ABB RAPID module: Module1.mod

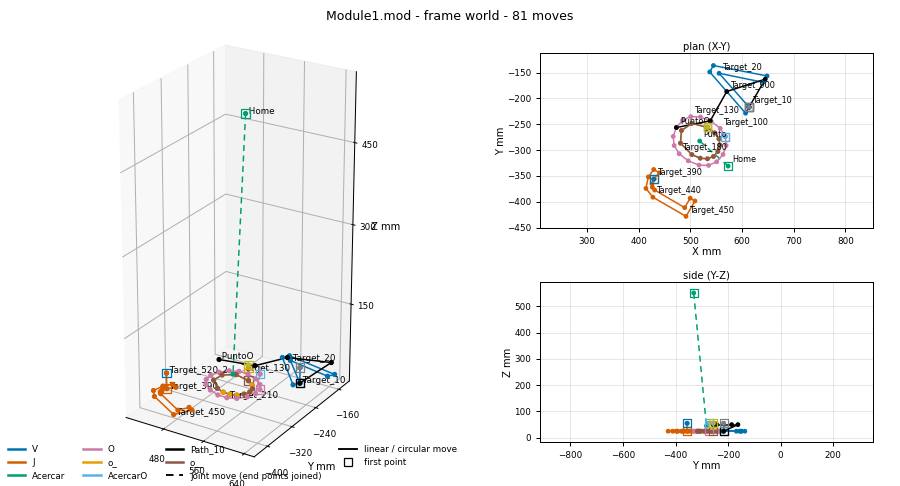
[picture p0: tool path of Module1.mod in frame world, 81 of 82 moves have a stored position in this frame; points joined in program order, loops and branches not executed]
MODULE Module1
        CONST robtarget Target_10:=[[139.847323193,319.022708542,15],[0,0.707106781,0.707106781,0],[0,0,0,0],[9E+09,9E+09,9E+09,9E+09,9E+09,9E+09]];
    CONST robtarget Target_20:=[[56.784114117,346.737457327,15],[0,0.707106781,0.707106781,0],[0,0,0,0],[9E+09,9E+09,9E+09,9E+09,9E+09,9E+09]];
    CONST robtarget Target_30:=[[139.847323193,374.452206111,15],[0,0.707106781,0.707106781,0],[0,0,0,0],[9E+09,9E+09,9E+09,9E+09,9E+09,9E+09]];
    CONST robtarget Target_40:=[[139.847323193,388.714766889,15],[0,0.707106781,0.707106781,0],[0,0,0,0],[9E+09,9E+09,9E+09,9E+09,9E+09,9E+09]];
    CONST robtarget Target_50:=[[39.847323193,354.273924101,15],[0,0.707106781,0.707106781,0],[0,0,0,0],[9E+09,9E+09,9E+09,9E+09,9E+09,9E+09]];
    CONST robtarget Target_60:=[[39.847323193,339.930326046,15],[0,0.707106781,0.707106781,0],[0,0,0,0],[9E+09,9E+09,9E+09,9E+09,9E+09,9E+09]];
    CONST robtarget Target_70:=[[139.847323193,305.489483258,15],[0,0.707106781,0.707106781,0],[0,0,0,0],[9E+09,9E+09,9E+09,9E+09,9E+09,9E+09]];
    CONST robtarget Target_80:=[[139.847323193,319.022708542,15],[0,0.707106781,0.707106781,0],[0,0,0,0],[9E+09,9E+09,9E+09,9E+09,9E+09,9E+09]];
    CONST robtarget Target_90:=[[128.421067116,246.656420049,15],[0,0.707106781,0.707106781,0],[0,0,0,0],[9E+09,9E+09,9E+09,9E+09,9E+09,9E+09]];
    CONST robtarget Target_100:=[[111.970499855,255.530001897,15],[0,0.707106781,0.707106781,0],[0,0,0,0],[9E+09,9E+09,9E+09,9E+09,9E+09,9E+09]];
    CONST robtarget Target_110:=[[89.847323193,258.649937067,15],[0,0.707106781,0.707106781,0],[0,0,0,0],[9E+09,9E+09,9E+09,9E+09,9E+09,9E+09]];
    CONST robtarget Target_120:=[[67.764665171,255.570520536,15],[0,0.707106781,0.707106781,0],[0,0,0,0],[9E+09,9E+09,9E+09,9E+09,9E+09,9E+09]];
    CONST robtarget Target_130:=[[51.354616548,246.737457327,15],[0,0.707106781,0.707106781,0],[0,0,0,0],[9E+09,9E+09,9E+09,9E+09,9E+09,9E+09]];
    CONST robtarget Target_140:=[[41.184438266,232.71800838,15],[0,0.707106781,0.707106781,0],[0,0,0,0],[9E+09,9E+09,9E+09,9E+09,9E+09,9E+09]];
    CONST robtarget Target_150:=[[37.740353988,214.484621022,15],[0,0.707106781,0.707106781,0],[0,0,0,0],[9E+09,9E+09,9E+09,9E+09,9E+09,9E+09]];
    CONST robtarget Target_460:=[[139.847323193,109.460309839,15],[0,0.707106781,0.707106781,0],[0,0,0,0],[9E+09,9E+09,9E+09,9E+09,9E+09,9E+09]];
    CONST robtarget Target_470:=[[129.231439887,109.460309839,15],[0,0.707106781,0.707106781,0],[0,0,0,0],[9E+09,9E+09,9E+09,9E+09,9E+09,9E+09]];
    CONST robtarget Target_480:=[[129.231439887,88.309580503,15],[0,0.707106781,0.707106781,0],[0,0,0,0],[9E+09,9E+09,9E+09,9E+09,9E+09,9E+09]];
    CONST robtarget Target_490:=[[61.970499855,88.795804166,15],[0,0.707106781,0.707106781,0],[0,0,0,0],[9E+09,9E+09,9E+09,9E+09,9E+09,9E+09]];
    CONST robtarget Target_500:=[[55.406480406,91.145885203,15],[0,0.707106781,0.707106781,0],[0,0,0,0],[9E+09,9E+09,9E+09,9E+09,9E+09,9E+09]];
    CONST robtarget Target_510:=[[51.395135187,96.534864134,15],[0,0.707106781,0.707106781,0],[0,0,0,0],[9E+09,9E+09,9E+09,9E+09,9E+09,9E+09]];
    CONST robtarget Target_520:=[[49.976982837,106.380893307,15],[0,0.707106781,0.707106781,0],[0,0,0,0],[9E+09,9E+09,9E+09,9E+09,9E+09,9E+09]];
    CONST robtarget Target_530:=[[129.231439887,88.309580503,15],[0,1,0,0],[0,0,0,0],[9E+09,9E+09,9E+09,9E+09,9E+09,9E+09]];
    CONST robtarget Target_540:=[[61.970499855,88.795804166,15],[0,1,0,0],[0,0,0,0],[9E+09,9E+09,9E+09,9E+09,9E+09,9E+09]];
    CONST robtarget Target_550:=[[55.406480406,91.145885203,15],[0,1,0,0],[0,0,0,0],[9E+09,9E+09,9E+09,9E+09,9E+09,9E+09]];
    CONST robtarget Target_560:=[[51.395135187,96.534864134,15],[0,1,0,0],[0,0,0,0],[9E+09,9E+09,9E+09,9E+09,9E+09,9E+09]];
    CONST robtarget Target_570:=[[49.976982837,106.380893307,15],[0,1,0,0],[0,0,0,0],[9E+09,9E+09,9E+09,9E+09,9E+09,9E+09]];
    CONST robtarget Target_580:=[[53.218473923,122.264199628,15],[0,1,0,0],[0,0,0,0],[9E+09,9E+09,9E+09,9E+09,9E+09,9E+09]];
    CONST robtarget Target_590:=[[40.414584134,122.264199628,15],[0,1,0,0],[0,0,0,0],[9E+09,9E+09,9E+09,9E+09,9E+09,9E+09]];
    CONST robtarget Home:=[[161.779515601,200,541.048881024],[0.5,0,0.866025404,0],[0,0,0,0],[9E+09,9E+09,9E+09,9E+09,9E+09,9E+09]];
    CONST robtarget Punto:=[[89.89,214.443,35],[0,1,0,0],[0,0,-2,0],[9E+09,9E+09,9E+09,9E+09,9E+09,9E+09]];
    CONST robtarget Target_600:=[[37.740353988,214.484621022,15],[0,1,0,0],[0,0,0,0],[9E+09,9E+09,9E+09,9E+09,9E+09,9E+09]];
    CONST robtarget Target_610:=[[41.062882351,196.534864134,15],[0,1,0,0],[0,0,0,0],[9E+09,9E+09,9E+09,9E+09,9E+09,9E+09]];
    CONST robtarget Target_620:=[[51.354616548,182.231784717,15],[0,1,0,0],[0,0,0,0],[9E+09,9E+09,9E+09,9E+09,9E+09,9E+09]];
    CONST robtarget Target_630:=[[67.845702448,173.317684231,15],[0,1,0,0],[0,0,0,0],[9E+09,9E+09,9E+09,9E+09,9E+09,9E+09]];
    CONST robtarget Target_640:=[[89.847323193,170.238267699,15],[0,1,0,0],[0,0,0,0],[9E+09,9E+09,9E+09,9E+09,9E+09,9E+09]];
    CONST robtarget Target_650:=[[112.051537132,173.398721508,15],[0,1,0,0],[0,0,0,0],[9E+09,9E+09,9E+09,9E+09,9E+09,9E+09]];
    CONST robtarget Target_660:=[[128.421067116,182.231784717,15],[0,1,0,0],[0,0,0,0],[9E+09,9E+09,9E+09,9E+09,9E+09,9E+09]];
    CONST robtarget Target_670:=[[138.388652205,196.089159109,15],[0,1,0,0],[0,0,0,0],[9E+09,9E+09,9E+09,9E+09,9E+09,9E+09]];
    CONST robtarget Target_680:=[[141.954292399,214.484621022,15],[0,1,0,0],[0,0,0,0],[9E+09,9E+09,9E+09,9E+09,9E+09,9E+09]];
    CONST robtarget Target_690:=[[138.510208121,232.677489741,15],[0,1,0,0],[0,0,0,0],[9E+09,9E+09,9E+09,9E+09,9E+09,9E+09]];
    CONST robtarget Target_700:=[[128.421067116,246.656420049,15],[0,1,0,0],[0,0,0,0],[9E+09,9E+09,9E+09,9E+09,9E+09,9E+09]];
    CONST robtarget Target_710:=[[111.970499855,255.530001897,15],[0,1,0,0],[0,0,0,0],[9E+09,9E+09,9E+09,9E+09,9E+09,9E+09]];
    CONST robtarget Target_720:=[[89.847323193,258.649937067,15],[0,1,0,0],[0,0,0,0],[9E+09,9E+09,9E+09,9E+09,9E+09,9E+09]];
    CONST robtarget Target_730:=[[67.764665171,255.570520536,15],[0,1,0,0],[0,0,0,0],[9E+09,9E+09,9E+09,9E+09,9E+09,9E+09]];
    CONST robtarget Target_740:=[[51.354616548,246.737457327,15],[0,1,0,0],[0,0,0,0],[9E+09,9E+09,9E+09,9E+09,9E+09,9E+09]];
    CONST robtarget Target_750:=[[41.184438266,232.71800838,15],[0,1,0,0],[0,0,0,0],[9E+09,9E+09,9E+09,9E+09,9E+09,9E+09]];
    CONST robtarget Target_760:=[[37.740353988,214.484621022,15],[0,1,0,0],[0,0,0,0],[9E+09,9E+09,9E+09,9E+09,9E+09,9E+09]];
    CONST robtarget Target_770:=[[89.847323193,244.792562675,15],[0,1,0,0],[0,0,0,0],[9E+09,9E+09,9E+09,9E+09,9E+09,9E+09]];
    CONST robtarget Target_780:=[[107.27033778,242.685593469,15],[0,1,0,0],[0,0,0,0],[9E+09,9E+09,9E+09,9E+09,9E+09,9E+09]];
    CONST robtarget Target_790:=[[120.074227569,236.607797683,15],[0,1,0,0],[0,0,0,0],[9E+09,9E+09,9E+09,9E+09,9E+09,9E+09]];
    CONST robtarget Target_800:=[[127.934843453,227.04539898,15],[0,1,0,0],[0,0,0,0],[9E+09,9E+09,9E+09,9E+09,9E+09,9E+09]];
    CONST robtarget Target_810:=[[130.446999044,214.403583745,15],[0,1,0,0],[0,0,0,0],[9E+09,9E+09,9E+09,9E+09,9E+09,9E+09]];
    CONST robtarget Target_820:=[[127.853806176,201.842805787,15],[0,1,0,0],[0,0,0,0],[9E+09,9E+09,9E+09,9E+09,9E+09,9E+09]];
    CONST robtarget Target_830:=[[120.074227569,192.280407083,15],[0,1,0,0],[0,0,0,0],[9E+09,9E+09,9E+09,9E+09,9E+09,9E+09]];
    CONST robtarget Target_840:=[[107.391893696,186.243129936,15],[0,1,0,0],[0,0,0,0],[9E+09,9E+09,9E+09,9E+09,9E+09,9E+09]];
    CONST robtarget Target_850:=[[89.847323193,184.095642092,15],[0,1,0,0],[0,0,0,0],[9E+09,9E+09,9E+09,9E+09,9E+09,9E+09]];
    CONST robtarget Target_860:=[[59.701456095,192.320925722,15],[0,1,0,0],[0,0,0,0],[9E+09,9E+09,9E+09,9E+09,9E+09,9E+09]];
    CONST robtarget Target_870:=[[49.247647343,214.403583745,15],[0,1,0,0],[0,0,0,0],[9E+09,9E+09,9E+09,9E+09,9E+09,9E+09]];
    CONST robtarget Target_880:=[[59.701456095,236.526760406,15],[0,1,0,0],[0,0,0,0],[9E+09,9E+09,9E+09,9E+09,9E+09,9E+09]];
    CONST robtarget Target_890:=[[89.847323193,244.792562675,15],[0,1,0,0],[0,0,0,0],[9E+09,9E+09,9E+09,9E+09,9E+09,9E+09]];
    CONST robtarget puntoV:=[[139.847,381.583,40],[0,1,0,0],[0,0,-2,0],[9E+09,9E+09,9E+09,9E+09,9E+09,9E+09]];
    CONST robtarget puntoV_2:=[[139.847,381.583,40],[0,1,0,0],[0,0,-2,0],[9E+09,9E+09,9E+09,9E+09,9E+09,9E+09]];
    CONST robtarget puntoJ_2:=[[40.415,122.264,40],[0,1,0,0],[-1,0,1,0],[9E+09,9E+09,9E+09,9E+09,9E+09,9E+09]];
    CONST robtarget puntoJ:=[[40.415,122.264,40],[0,1,0,0],[-1,0,1,0],[9E+09,9E+09,9E+09,9E+09,9E+09,9E+09]];
    CONST robtarget PuntoO_2:=[[37.74,214.485,40],[0,1,0,0],[0,0,0,0],[9E+09,9E+09,9E+09,9E+09,9E+09,9E+09]];
    CONST robtarget PuntoO:=[[37.740005074,214.485004022,40.000022651],[0,1,0,0],[0,0,-2,0],[9E+09,9E+09,9E+09,9E+09,9E+09,9E+09]];
    CONST robtarget punto_opeq_2:=[[89.847,244.793,40],[0,1,0,0],[0,0,0,0],[9E+09,9E+09,9E+09,9E+09,9E+09,9E+09]];
    CONST robtarget punto_opeq:=[[89.847,244.793,40],[0,1,0,0],[0,0,0,0],[9E+09,9E+09,9E+09,9E+09,9E+09,9E+09]];
    CONST robtarget Target_900:=[[87.275,323.596,40],[0,1,0,0],[0,0,-2,0],[9E+09,9E+09,9E+09,9E+09,9E+09,9E+09]];
    CONST robtarget Target_910:=[[88.022,258.633,40],[0,1,0,0],[0,0,-2,0],[9E+09,9E+09,9E+09,9E+09,9E+09,9E+09]];
    CONST robtarget Target_80_2:=[[139.847323193,319.022708542,45],[0,0.707106781,0.707106781,0],[0,0,1,0],[9E+09,9E+09,9E+09,9E+09,9E+09,9E+09]];
    CONST robtarget Target_160:=[[41.062882351,196.534864134,15],[0,0.707106781,0.707106781,0],[0,0,0,0],[9E+09,9E+09,9E+09,9E+09,9E+09,9E+09]];
    CONST robtarget Target_230:=[[141.954292399,214.484621022,15],[0,0.707106781,0.707106781,0],[0,0,0,0],[9E+09,9E+09,9E+09,9E+09,9E+09,9E+09]];
    CONST robtarget Target_180:=[[67.845702448,173.317684231,15],[0,0.707106781,0.707106781,0],[0,0,0,0],[9E+09,9E+09,9E+09,9E+09,9E+09,9E+09]];
    CONST robtarget Target_240:=[[138.510208121,232.677489741,15],[0,0.707106781,0.707106781,0],[0,0,0,0],[9E+09,9E+09,9E+09,9E+09,9E+09,9E+09]];
    CONST robtarget Target_200:=[[112.051537132,173.398721508,15],[0,0.707106781,0.707106781,0],[0,0,0,0],[9E+09,9E+09,9E+09,9E+09,9E+09,9E+09]];
    CONST robtarget Target_220:=[[138.388652205,196.089159109,15],[0,0.707106781,0.707106781,0],[0,0,0,0],[9E+09,9E+09,9E+09,9E+09,9E+09,9E+09]];
    CONST robtarget Target_170:=[[51.354616548,182.231784717,15],[0,0.707106781,0.707106781,0],[0,0,0,0],[9E+09,9E+09,9E+09,9E+09,9E+09,9E+09]];
    CONST robtarget Target_210:=[[128.421067116,182.231784717,15],[0,0.707106781,0.707106781,0],[0,0,0,0],[9E+09,9E+09,9E+09,9E+09,9E+09,9E+09]];
    CONST robtarget Target_190:=[[89.847323193,170.238267699,15],[0,0.707106781,0.707106781,0],[0,0,0,0],[9E+09,9E+09,9E+09,9E+09,9E+09,9E+09]];
    CONST robtarget Target_250_2:=[[128.421067116,246.656420049,45],[0,0.707106781,0.707106781,0],[0,0,1,0],[9E+09,9E+09,9E+09,9E+09,9E+09,9E+09]];
    CONST robtarget Target_260:=[[89.847323193,244.792562675,15],[0,0.707106781,0.707106781,0],[0,0,0,0],[9E+09,9E+09,9E+09,9E+09,9E+09,9E+09]];
    CONST robtarget Target_270:=[[107.27033778,242.685593469,15],[0,0.707106781,0.707106781,0],[0,0,0,0],[9E+09,9E+09,9E+09,9E+09,9E+09,9E+09]];
    CONST robtarget Target_280:=[[120.074227569,236.607797683,15],[0,0.707106781,0.707106781,0],[0,0,0,0],[9E+09,9E+09,9E+09,9E+09,9E+09,9E+09]];
    CONST robtarget Target_290:=[[127.934843453,227.04539898,15],[0,0.707106781,0.707106781,0],[0,0,0,0],[9E+09,9E+09,9E+09,9E+09,9E+09,9E+09]];
    CONST robtarget Target_300:=[[130.446999044,214.403583745,15],[0,0.707106781,0.707106781,0],[0,0,0,0],[9E+09,9E+09,9E+09,9E+09,9E+09,9E+09]];
    CONST robtarget Target_310:=[[127.853806176,201.842805787,15],[0,0.707106781,0.707106781,0],[0,0,0,0],[9E+09,9E+09,9E+09,9E+09,9E+09,9E+09]];
    CONST robtarget Target_320:=[[120.074227569,192.280407083,15],[0,0.707106781,0.707106781,0],[0,0,0,0],[9E+09,9E+09,9E+09,9E+09,9E+09,9E+09]];
    CONST robtarget Target_330:=[[107.391893696,186.243129936,15],[0,0.707106781,0.707106781,0],[0,0,0,0],[9E+09,9E+09,9E+09,9E+09,9E+09,9E+09]];
    CONST robtarget Target_340:=[[89.847323193,184.095642092,15],[0,0.707106781,0.707106781,0],[0,0,0,0],[9E+09,9E+09,9E+09,9E+09,9E+09,9E+09]];
    CONST robtarget Target_350:=[[59.701456095,192.320925722,15],[0,0.707106781,0.707106781,0],[0,0,0,0],[9E+09,9E+09,9E+09,9E+09,9E+09,9E+09]];
    CONST robtarget Target_360:=[[49.247647343,214.403583745,15],[0,0.707106781,0.707106781,0],[0,0,0,0],[9E+09,9E+09,9E+09,9E+09,9E+09,9E+09]];
    CONST robtarget Target_370:=[[59.701456095,236.526760406,15],[0,0.707106781,0.707106781,0],[0,0,0,0],[9E+09,9E+09,9E+09,9E+09,9E+09,9E+09]];
    CONST robtarget Target_380:=[[89.847323193,244.792562675,15],[0,0.707106781,0.707106781,0],[0,0,0,0],[9E+09,9E+09,9E+09,9E+09,9E+09,9E+09]];
    CONST robtarget Target_380_2:=[[89.847323193,244.792562675,45],[0,0.707106781,0.707106781,0],[0,0,1,0],[9E+09,9E+09,9E+09,9E+09,9E+09,9E+09]];
    CONST robtarget Target_520_2:=[[49.976982837,106.380893307,45],[0,0.707106781,0.707106781,0],[0,0,0,0],[9E+09,9E+09,9E+09,9E+09,9E+09,9E+09]];
    CONST robtarget Target_410:=[[40.414584134,122.264199628,15],[0,0.707106781,0.707106781,0],[0,0,0,0],[9E+09,9E+09,9E+09,9E+09,9E+09,9E+09]];
    CONST robtarget Target_400:=[[53.218473923,122.264199628,15],[0,0.707106781,0.707106781,0],[0,0,0,0],[9E+09,9E+09,9E+09,9E+09,9E+09,9E+09]];
    CONST robtarget Target_390:=[[49.976982837,106.380893307,15],[0,0.707106781,0.707106781,0],[0,0,0,0],[9E+09,9E+09,9E+09,9E+09,9E+09,9E+09]];
    CONST robtarget Target_440:=[[65.860289158,75.019467051,15],[0,0.707106781,0.707106781,0],[0,0,0,0],[9E+09,9E+09,9E+09,9E+09,9E+09,9E+09]];
    CONST robtarget Target_420:=[[38.469689482,104.59807321,15],[0,0.707106781,0.707106781,0],[0,0,0,0],[9E+09,9E+09,9E+09,9E+09,9E+09,9E+09]];
    CONST robtarget Target_430:=[[45.600969871,83.042157489,15],[0,0.707106781,0.707106781,0],[0,0,0,0],[9E+09,9E+09,9E+09,9E+09,9E+09,9E+09]];
    CONST robtarget Target_450:=[[139.847323193,75.019467051,15],[0,0.707106781,0.707106781,0],[0,0,0,0],[9E+09,9E+09,9E+09,9E+09,9E+09,9E+09]];
    CONST jointtarget home2:=[[0,0,0,0,0,0],[9E+09,9E+09,9E+09,9E+09,9E+09,9E+09]];
!***********************************************************
    !
    ! Module:  Module1
    !
    ! Description:
    !   <Insert description here>
    !
    ! Author: Valentina Cruz DP
    !
    ! Version: 1.0
    !
    !***********************************************************


    !***********************************************************
    !
    ! Procedure main
    !
    !   This is the entry point of your program
    !
    !***********************************************************
    PROC main()

     homee;
     AcercarV;
     V;
     AcercarO;
     O;
     AcercarO_;
     o__;
     AcercarJ;
     J;
     homee;

    ENDPROC
    PROC V()
        MoveL Target_10,v60,z1,HerramientaVOJ\WObj:=WorkobjectVOJ;
        MoveL Target_20,v60,z1,HerramientaVOJ\WObj:=WorkobjectVOJ;
        MoveL Target_30,v60,z1,HerramientaVOJ\WObj:=WorkobjectVOJ;
        MoveL Target_40,v60,z1,HerramientaVOJ\WObj:=WorkobjectVOJ;
        MoveL Target_50,v60,z1,HerramientaVOJ\WObj:=WorkobjectVOJ;
        MoveL Target_60,v60,z1,HerramientaVOJ\WObj:=WorkobjectVOJ;
        MoveL Target_70,v60,z1,HerramientaVOJ\WObj:=WorkobjectVOJ;
        MoveL Target_80,v60,z1,HerramientaVOJ\WObj:=WorkobjectVOJ;
        MoveL Target_80_2,v60,z1,HerramientaVOJ\WObj:=WorkobjectVOJ;
    ENDPROC
    PROC J()
        MoveL Target_390,v60,z1,HerramientaVOJ\WObj:=WorkobjectVOJ;
        MoveL Target_400,v60,z1,HerramientaVOJ\WObj:=WorkobjectVOJ;
        MoveL Target_410,v60,z1,HerramientaVOJ\WObj:=WorkobjectVOJ;
        MoveL Target_420,v60,z1,HerramientaVOJ\WObj:=WorkobjectVOJ;
        MoveL Target_430,v60,z1,HerramientaVOJ\WObj:=WorkobjectVOJ;
        MoveL Target_440,v60,z1,HerramientaVOJ\WObj:=WorkobjectVOJ;
        MoveL Target_450,v60,z1,HerramientaVOJ\WObj:=WorkobjectVOJ;
        MoveL Target_460,v60,z1,HerramientaVOJ\WObj:=WorkobjectVOJ;
        MoveL Target_470,v60,z1,HerramientaVOJ\WObj:=WorkobjectVOJ;
        MoveL Target_480,v60,z1,HerramientaVOJ\WObj:=WorkobjectVOJ;
        MoveL Target_490,v60,z1,HerramientaVOJ\WObj:=WorkobjectVOJ;
        MoveL Target_500,v60,z1,HerramientaVOJ\WObj:=WorkobjectVOJ;
        MoveL Target_510,v60,z1,HerramientaVOJ\WObj:=WorkobjectVOJ;
        MoveL Target_520,v60,z1,HerramientaVOJ\WObj:=WorkobjectVOJ;
        MoveL Target_520_2,v60,z1,HerramientaVOJ\WObj:=WorkobjectVOJ;
    ENDPROC
    PROC Acercar()
        MoveJ Home,v200,z1,HerramientaVOJ\WObj:=WorkobjectVOJ;
        MoveJ Punto,v200,z1,HerramientaVOJ\WObj:=WorkobjectVOJ;
    ENDPROC
    PROC Alejar()
    ENDPROC
    PROC O()
        MoveL Target_90,v60,z1,HerramientaVOJ\WObj:=WorkobjectVOJ;
        MoveL Target_100,v60,z1,HerramientaVOJ\WObj:=WorkobjectVOJ;
        MoveL Target_110,v60,z1,HerramientaVOJ\WObj:=WorkobjectVOJ;
        MoveL Target_120,v60,z1,HerramientaVOJ\WObj:=WorkobjectVOJ;
        MoveL Target_130,v60,z1,HerramientaVOJ\WObj:=WorkobjectVOJ;
        MoveL Target_140,v60,z1,HerramientaVOJ\WObj:=WorkobjectVOJ;
        MoveL Target_150,v60,z1,HerramientaVOJ\WObj:=WorkobjectVOJ;
        MoveL Target_160,v60,z1,HerramientaVOJ\WObj:=WorkobjectVOJ;
        MoveL Target_170,v60,z1,HerramientaVOJ\WObj:=WorkobjectVOJ;
        MoveL Target_180,v60,z1,HerramientaVOJ\WObj:=WorkobjectVOJ;
        MoveL Target_190,v60,z1,HerramientaVOJ\WObj:=WorkobjectVOJ;
        MoveL Target_200,v60,z1,HerramientaVOJ\WObj:=WorkobjectVOJ;
        MoveL Target_210,v60,z1,HerramientaVOJ\WObj:=WorkobjectVOJ;
        MoveL Target_220,v60,z1,HerramientaVOJ\WObj:=WorkobjectVOJ;
        MoveL Target_230,v60,z1,HerramientaVOJ\WObj:=WorkobjectVOJ;
        MoveL Target_240,v60,z1,HerramientaVOJ\WObj:=WorkobjectVOJ;
        MoveL Target_250_2,v60,z1,HerramientaVOJ\WObj:=WorkobjectVOJ;
    ENDPROC
    PROC o_()
        MoveL punto_opeq_2,v60,z1,HerramientaVOJ\WObj:=WorkobjectVOJ;
        MoveL Target_770,v60,z1,HerramientaVOJ\WObj:=WorkobjectVOJ;
        MoveL Target_780,v60,z1,HerramientaVOJ\WObj:=WorkobjectVOJ;
        MoveL Target_790,v60,z1,HerramientaVOJ\WObj:=WorkobjectVOJ;
        MoveL Target_800,v60,z1,HerramientaVOJ\WObj:=WorkobjectVOJ;
        MoveL Target_810,v60,z1,HerramientaVOJ\WObj:=WorkobjectVOJ;
        MoveL Target_820,v60,z1,HerramientaVOJ\WObj:=WorkobjectVOJ;
        MoveL Target_830,v60,z1,HerramientaVOJ\WObj:=WorkobjectVOJ;
        MoveL Target_840,v60,z1,HerramientaVOJ\WObj:=WorkobjectVOJ;
        MoveL Target_850,v60,z1,HerramientaVOJ\WObj:=WorkobjectVOJ;
        MoveL Target_860,v60,z1,HerramientaVOJ\WObj:=WorkobjectVOJ;
        MoveL Target_870,v60,z1,HerramientaVOJ\WObj:=WorkobjectVOJ;
        MoveL Target_880,v60,z1,HerramientaVOJ\WObj:=WorkobjectVOJ;
        MoveL Target_890,v60,z1,HerramientaVOJ\WObj:=WorkobjectVOJ;
        MoveL punto_opeq,v60,z1,HerramientaVOJ\WObj:=WorkobjectVOJ;
    ENDPROC
    PROC AcercarO()
        MoveJ Target_250_2,v60,z1,HerramientaVOJ\WObj:=WorkobjectVOJ;
    ENDPROC
    PROC Path_10()
        MoveL Target_10,v200,z1,HerramientaVOJ\WObj:=WorkobjectVOJ;
        MoveL puntoV,v200,z1,HerramientaVOJ\WObj:=WorkobjectVOJ;
        MoveL Target_900,v200,z1,HerramientaVOJ\WObj:=WorkobjectVOJ;
        MoveL Target_910,v200,z1,HerramientaVOJ\WObj:=WorkobjectVOJ;
        MoveL PuntoO,v200,z1,HerramientaVOJ\WObj:=WorkobjectVOJ;
    ENDPROC
    PROC o__()
        MoveL Target_260,v60,z1,HerramientaVOJ\WObj:=WorkobjectVOJ;
        MoveL Target_270,v60,z1,HerramientaVOJ\WObj:=WorkobjectVOJ;
        MoveL Target_280,v60,z1,HerramientaVOJ\WObj:=WorkobjectVOJ;
        MoveL Target_290,v60,z1,HerramientaVOJ\WObj:=WorkobjectVOJ;
        MoveL Target_300,v60,z1,HerramientaVOJ\WObj:=WorkobjectVOJ;
        MoveL Target_310,v60,z1,HerramientaVOJ\WObj:=WorkobjectVOJ;
        MoveL Target_320,v60,z1,HerramientaVOJ\WObj:=WorkobjectVOJ;
        MoveL Target_330,v60,z1,HerramientaVOJ\WObj:=WorkobjectVOJ;
        MoveL Target_340,v60,z1,HerramientaVOJ\WObj:=WorkobjectVOJ;
        MoveL Target_350,v60,z1,HerramientaVOJ\WObj:=WorkobjectVOJ;
        MoveL Target_360,v60,z1,HerramientaVOJ\WObj:=WorkobjectVOJ;
        MoveL Target_370,v60,z1,HerramientaVOJ\WObj:=WorkobjectVOJ;
        MoveL Target_380,v60,z1,HerramientaVOJ\WObj:=WorkobjectVOJ;
        MoveL Target_380_2,v60,z1,HerramientaVOJ\WObj:=WorkobjectVOJ;
    ENDPROC
    PROC AcercarV()
        MoveJ Target_80_2,v60,z1,HerramientaVOJ\WObj:=WorkobjectVOJ;
    ENDPROC
    PROC AcercarO_()
        MoveJ Target_380_2,v60,z1,HerramientaVOJ\WObj:=WorkobjectVOJ;
    ENDPROC
    PROC AcercarJ()
        MoveJ Target_520_2,v60,z1,HerramientaVOJ\WObj:=WorkobjectVOJ;
    ENDPROC
    PROC homee()
        MoveAbsJ home2,v1000,z100,HerramientaVOJ\WObj:=g;
    ENDPROC
ENDMODULE
